FUNCTION A_REAL : ST_Arg
VAR_INPUT
	fNumber	: REFERENCE TO REAL;
END_VAR

IF __ISVALIDREF(fNumber) THEN
	A_REAL.eType := E_ArgType.RealArg;
	A_REAL.pData := ADR(fNumber);
	A_REAL.nSize := SIZEOF(REAL);
END_IF

END_FUNCTION

(* stored: Version 1.1.0.1, ProductVersion 3.1.4024.15
   POU A_REAL: Id {037dc33e-6fe3-4fa2-8c95-f9a85fea31d9}, SpecialFunc None *)
